FUNCTION_BLOCK fb_Process_LinkedListCtrl IMPLEMENTS I_Process_LinkedList
VAR
  _LastNodeAdded,
  _LastNodeRemoved  : ST_PROCESS_LIST_RESULT;

	_nCount           : UDINT;
  _nFree            : UDINT;

  {attribute 'hide'}
	_stList           : ARRAY[0..MAX_LIST_NODES] OF ST_PROCESS_DATA;
	_stNodes          : ARRAY[0..MAX_LIST_NODES] OF T_LinkedListEntry;

	_fbList           : Tc2_Utilities.FB_LinkedListCtrl;
	_hList            : Tc2_Utilities.T_HLINKEDLIST;

	_stRef            : POINTER TO ST_PROCESS_DATA;
END_VAR

METHOD AddHeadValue : ST_PROCESS_LIST_RESULT
VAR_INPUT
  stData        : ST_PROCESS_DATA;
END_VAR
VAR
  _nIdxNode     : ULINT; 
	_pPosGet      : POINTER TO T_LinkedListEntry;
  _stRes        : ST_PROCESS_LIST_RESULT;
END_VAR

// add empty node
_fbList.A_AddHeadValue( hList     := _hList, 
                        putValue  := 16#0, 
                        getPosPtr => _pPosGet);

IF NOT _fbList.bOk 
THEN
  _stRes.wState.0       := TRUE;
ELSE
  // Get array index of new node
	_fbList.A_GetIndexAtPosPtr( hList       := _hList, 
                              putPosPtr   := _pPosGet, 
                              getValue    => _nIdxNode);

	IF NOT _fbList.bOk 
  THEN
    _stRes.wState.1     := TRUE;
  ELSE
    // write data to new node index
		_stRef 	            := ADR( _stList[_nIdxNode] );
		_stRef^ 	          := stData;

		_fbList.A_SetValueAtPosPtr( hList     := _hList, 
                                putPosPtr := _pPosGet, 
                                putValue  := _stRef);

		IF NOT _fbList.bOk 
    THEN
      _stRes.wState.2   := TRUE;
    ELSE
      _stRes.nIndex     := _nIdxNode;
			_stRes.stData     := stData;
      _LastNodeAdded    := _stRes;
		END_IF
	END_IF
END_IF
_nCount       := _hList.nCount;
_nFree        := _hList.nFree;
AddHeadValue  := _stRes;
END_METHOD

METHOD AddTailValue : ST_PROCESS_LIST_RESULT
VAR_INPUT
  stData        : ST_PROCESS_DATA;
END_VAR
VAR
  _nIdxNode     : ULINT; 
	_pPosGet      : POINTER TO T_LinkedListEntry;
  _stRes        : ST_PROCESS_LIST_RESULT;
END_VAR

// add empty node
_fbList.A_AddTailValue( hList       := _hList, 
                        putValue    := 16#0, 
                        getPosPtr   => _pPosGet);


IF NOT _fbList.bOk 
THEN
  _stRes.wState.0 := TRUE;
ELSE
  // Get array index of new node
	_fbList.A_GetIndexAtPosPtr( hList       := _hList, 
                              putPosPtr   := _pPosGet, 
                              getValue    => _nIdxNode);

	IF NOT _fbList.bOk 
  THEN
    _stRes.wState.1     := TRUE;
  ELSE
    // write data to new node index
		_stRef 	            := ADR( _stList[_nIdxNode] );
		_stRef^ 	          := stData;

		_fbList.A_SetValueAtPosPtr( hList     := _hList, 
                                putPosPtr := _pPosGet, 
                                putValue  := _stRef);

		IF NOT _fbList.bOk 
    THEN
      _stRes.wState.2   := TRUE;
    ELSE
      _stRes.nIndex     := _nIdxNode;
			_stRes.stData     := stData;
      _LastNodeAdded    := _stRes;
		END_IF
	END_IF
END_IF
_nCount       := _hList.nCount;
_nFree        := _hList.nFree;
AddTailValue  := _stRes;
END_METHOD

PROPERTY Count : UDINT
GET
Count := _nCount := _hList.nCount;
END_GET
END_PROPERTY

PROPERTY Data : ARRAY[1..MAX_LIST_NODES] OF ST_PROCESS_DATA
GET
VAR
	_tList        : ARRAY[1..MAX_LIST_NODES] OF ST_PROCESS_DATA;
  _getValue     : PVOID;
  _pEntry       : POINTER TO ST_PROCESS_DATA;
  _getPosPtr    : POINTER TO T_LinkedListEntry := 0;
  _nIdx         : UINT;  
END_VAR
_fbList(
	hList       := _hList);

_nCount       := _hList.nCount;
_nFree        := _hList.nFree;


_fbList.A_GetHead( hList := _hList, getValue=> _getValue, getPosPtr=> _getPosPtr );
IF _fbList.bOk 
THEN
  IF (_hList.nCount > 0)
  THEN
    _nIdx         := 1;
    _pEntry       := _getValue;
    _tList[1]     := _pEntry^;
    
    REPEAT
      _fbList.A_GetNext( hList := _hList, putPosPtr := _getPosPtr, getValue=> _getValue, getPosPtr=> _getPosPtr );
  
      IF _fbList.bOk THEN
        _nIdx         := _nIdx + 1;
        _pEntry       := _getValue;
        _tList[_nIdx] := _pEntry^;
      ELSE
        EXIT;
      END_IF
    UNTIL NOT _fbList.bOk
    END_REPEAT
  END_IF
END_IF

Data := _tList;
END_GET
END_PROPERTY

PROPERTY Free : UDINT
GET
Free := _nFree := _hList.nFree;
END_GET
END_PROPERTY

METHOD GetHead : ST_PROCESS_LIST_RESULT
VAR_INPUT
END_VAR
VAR
	_pPosGet      : POINTER TO T_LinkedListEntry;
  _pData        : POINTER TO ST_PROCESS_DATA;
  _stRes        : ST_PROCESS_LIST_RESULT;
END_VAR

_fbList.A_GetHead(hList      := _hList,
                  getValue   => _pData,
                  getPosPtr  => _pPosGet);

IF NOT _fbList.bOk
THEN
  _stRes.wState.0 := TRUE;
ELSE
  _stRes.stData := _pData^;
END_IF
_nCount       := _hList.nCount;
_nFree        := _hList.nFree;
GetHead       := _stRes;
END_METHOD

METHOD GetTail : ST_PROCESS_LIST_RESULT
VAR_INPUT
END_VAR
VAR
	_pPosGet      : POINTER TO T_LinkedListEntry;
  _pData        : POINTER TO ST_PROCESS_DATA;
  _stRes        : ST_PROCESS_LIST_RESULT;
END_VAR

_fbList.A_GetTail(hList      := _hList,
                  getValue   => _pData,
                  getPosPtr  => _pPosGet);

IF NOT _fbList.bOk
THEN
  _stRes.wState.0 := TRUE;
ELSE
  _stRes.stData := _pData^;
END_IF
_nCount       := _hList.nCount;
_nFree        := _hList.nFree;
GetTail       := _stRes;
END_METHOD

METHOD InitList : BOOL
VAR
  _bOk : Bool;
END_VAR

IF Tc2_Utilities.F_CreateLinkedListHnd(ADR(_stNodes), SIZEOF(_stNodes), _hList)
THEN
  _fbList.A_Reset(hList := _hList, bOk => _bOk);
  memset(ADR(_stList), 0, SIZEOF(_stList));
  _nCount   := _hList.nCount;
  _nFree    := _hList.nFree;
  InitList  := TRUE; //_bOk;
END_IF
END_METHOD

PROPERTY Nodes : ARRAY[0..MAX_LIST_NODES] OF T_LinkedListEntry
GET
Nodes := _stNodes;
END_GET
END_PROPERTY

METHOD RemoveHeadValue : ST_PROCESS_LIST_RESULT
VAR_INPUT
END_VAR
VAR
	_pPosGet      : POINTER TO T_LinkedListEntry;
  _pData        : POINTER TO ST_PROCESS_DATA;
  _stRes        : ST_PROCESS_LIST_RESULT;
END_VAR
_fbList.A_RemoveHeadValue(hList       := _hList, 
                          getValue    => _pData, 
                          getPosPtr   => _pPosGet);

IF NOT _fbList.bOk 
THEN
  _stRes.wState.0 := TRUE;
ELSE
	_stRes.stData     := _pData^;
  _LastNodeRemoved  := _stRes;
  memset(_pData, 0, SIZEOF(ST_PROCESS_DATA));
END_IF
_nCount           := _hList.nCount;
_nFree            := _hList.nFree;
RemoveHeadValue   := _stRes;
END_METHOD

END_FUNCTION_BLOCK

(* stored: Version 1.1.0.1, ProductVersion 3.1.4024.15
   POU fb_Process_LinkedListCtrl: Id {d481acc0-8bbd-42d4-bc58-58db20d0c7e4}, SpecialFunc None
   Method AddHeadValue: Id {cb088eeb-ebce-4b55-9535-78faa263e675}
   Method AddTailValue: Id {4b36eae4-75f4-4e48-886d-a9b9d29a7cba}
   Property Count: Id {8ce88ace-6381-4814-9e6c-78dcc915ba31}
   Get Get: Id {05a72a22-76f7-4cce-8891-436b9915e4a6}
   Property Data: Id {04469e6f-0b47-4af8-9a80-285cec8de7dd}
   Get Get: Id {ac84b142-7e05-4c51-b3b9-9ecb2eb2fd21}
   Property Free: Id {7fcb031f-f413-4391-8997-07e7dea8e9db}
   Get Get: Id {d5a9f1ac-fb1b-4722-86a0-58426ae277ea}
   Method GetHead: Id {8b3b30bf-f6ca-46d8-98f5-aa9e88db4597}
   Method GetTail: Id {ee04005f-daf4-444d-a863-b6c4aa3ebce0}
   Method InitList: Id {d197dbd8-b906-4214-bb4b-a515f9ab5a7d}
   Property Nodes: Id {88cd6309-4ace-45b9-9128-9513c4912c72}
   Get Get: Id {09ab2d93-99d0-4583-9280-54d1d4d4964d}
   Method RemoveHeadValue: Id {0edf66db-7029-4462-af17-168d20a4430a} *)
